(* IEC 61131-3 sources: MyDemoProject/src, 2 files *)

(* ---- ItemCounter.st ---- *)
NAMESPACE Stan
    // This class counts items
    CLASS PUBLIC ItemCounter
        VAR PROTECTED
            _value : DINT;
        END_VAR

        // Set CounterValue to value if value >0; If value <0 then CounterValue will be set to 0
        METHOD PUBLIC SetCounterValue
            VAR_INPUT
                value : DINT;
            END_VAR
            IF (value < 0) THEN
                _value := 0;
                RETURN;
            END_IF;
            _value := value;
        END_METHOD

        // Increase the counter by value 1
        METHOD PUBLIC CountItem
            _value := _value + DINT#1;
        END_METHOD

        // Returns the actual counter value
        METHOD PUBLIC GetCounterValue : DINT
            GetCounterValue := _value;
        END_METHOD
    END_CLASS
END_NAMESPACE

(* ---- itemCounterTiap.st ---- *)
NAMESPACE Stan.Standardizer

    FUNCTION_BLOCK ItemCounterTiap

        VAR_INPUT
            Execute : BOOL;
        END_VAR
        VAR_OUTPUT
            Counts : DINT;
            Message : STRING;
        END_VAR
        VAR
            _counter : ItemCounter;
            _executeOld : BOOL;
            _initDone : BOOL;
        END_VAR
        VAR_TEMP
            tempExecuteRis : BOOL;
        END_VAR

        tempExecuteRis := Execute AND NOT _executeOld;
        _executeOld := Execute;

        IF(NOT(_initDone)) THEN
            // Message := counter.toString();
            _initDone := true;
        END_IF;
        IF(tempExecuteRis) THEN
            _counter.CountItem();
            Counts := _counter.GetCounterValue();
            // Message := _counter.ToString();
        END_IF;

    END_FUNCTION_BLOCK

END_NAMESPACE
